FUNCTION_BLOCK FB_CamOut_Empty
VAR_INPUT
  Slave             : REFERENCE TO Tc2_MC2.AXIS_REF;
  Execute           : BOOL;
END_VAR
VAR_OUTPUT
  Busy              : BOOL;
  Error             : BOOL;
  Done              : BOOL;
  ErrorId           : UDINT;
END_VAR
VAR
END_VAR


Error   := TRUE;
ErrorId := 9999; // function is not activated by compiler def CAM

END_FUNCTION_BLOCK

(* stored: Version 1.1.0.1, ProductVersion 3.1.4024.9
   POU FB_CamOut_Empty: Id {cd80eb01-b0e2-0e5b-0b55-ab0c52f95ff7}, SpecialFunc None *)
